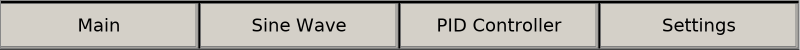
VISUALIZATION TogelSwich  // 800x50
    Rectangle (-1,1 800x50)
    Button (400,3 198x45), "PID Controller"
        OnMouseDown: change screen: Screen_PID_Control
    Button (0,3 198x45), "Main"
        OnMouseDown: change screen: Main_screen
    Button (200,3 198x45), "Sine Wave"
        OnMouseDown: change screen: Visualization
    Button (600,3 198x45), "Settings"
        OnMouseDown: change screen: Settings
END_VISUALIZATION

(* stored: Version 1.1.0.1, ProductVersion 3.1.4024.12
   Visu TogelSwich: Id {91899231-7726-4060-b203-eb49296b54c8} *)
